Staubli VAL3: pick.pgx

program pick(num x_nX, num x_nY, num x_angle, tool tGreifer)
  local num i
begin

  i = 0


  switch nData[0]

    case 1
      if nData[1] == 1
        i = 1
      endIf

    break
    case 2
      if nData[1] == 1
        i = 3
      else
        i = 2
      endIf


    break
    default
      i = 1
    break
  endSwitch

  //logMsg("n_Y "+toString(".4",x_nY))
  //logMsg("i: " + toString("0.4",i))
  pPick[i].trsf.x = x_nX
  pPick[i].trsf.y = x_nY
  pPick[i].trsf.rz = x_angle



  movej(appro(pPick[i],trApro),tGreifer, mUsedSpeed)
  movel(pPick[i], tGreifer, mUsedSpeed)
  close(tGreifer)
  movel(appro(pPick[i], trApro), tGreifer, mUsedSpeed)
  //logMsg("Objekt aufgegriffen")







end
